  def rq_gripper_led_force_blue(gripper_socket="1"):
      rq_set_var(LBP,1, gripper_socket)
      rq_set_var(LRD,0, gripper_socket)
      rq_set_var(LBL,1, gripper_socket)
      rq_set_var(LGN,0, gripper_socket)
  end

  def rq_gripper_led_force_green(gripper_socket="1"):
      rq_set_var(LBP,1, gripper_socket)
      rq_set_var(LRD,0, gripper_socket)
      rq_set_var(LBL,0, gripper_socket)
      rq_set_var(LGN,1, gripper_socket)
  end

  def rq_gripper_led_force_purple(gripper_socket="1"):
      rq_set_var(LBP,1, gripper_socket)
      rq_set_var(LRD,1, gripper_socket)
      rq_set_var(LBL,1, gripper_socket)
      rq_set_var(LGN,0, gripper_socket)
  end

  ############################################
  # mm/inches functions
  ############################################
  gripper_closed_norm = [100, 100, 100, 100]
  gripper_open_norm = [0, 0, 0, 0]
  gripper_closed_mm = [0, 0, 0, 0]
  gripper_open_mm = [50, 50, 50, 50]

  def rq_current_pos_mm(gripper_socket=1):
      pos_gripper = rq_current_pos(gripper_socket)
      pos_mm = gripper_to_mm(pos_gripper, gripper_socket)
      return round_value_2_dec(pos_mm)
  end

  def rq_current_pos_inches(gripper_socket=1):
      pos_gripper = rq_current_pos(gripper_socket)
      pos_mm = gripper_to_mm(pos_gripper, gripper_socket)
      pos_in = pos_mm / 25.4
      return round_value_2_dec(pos_in)
  end

  def rq_move_mm(pos_mm, gripper_socket=1):
      pos_gripper = mm_to_gripper(pos_mm, gripper_socket)
      rq_move(pos_gripper, gripper_socket)
  end

  def rq_move_and_wait_mm(pos_mm, gripper_socket=1):
      pos_gripper = mm_to_gripper(pos_mm, gripper_socket)
      rq_move_and_wait(pos_gripper, gripper_socket)
  end

  def rq_move_inches(pos_in, gripper_socket=1):
      pos_mm = pos_in * 25.4
      rq_move_mm(pos_mm, gripper_socket)
  end

  def rq_move_and_wait_inches(pos_in, gripper_socket=1):
      pos_mm = pos_in * 25.4
      rq_move_and_wait_mm(pos_mm, gripper_socket)
  end

  def get_closed_norm(gripper_socket):
      return gripper_closed_norm[gripper_socket - 1]
  end

  def get_open_norm(gripper_socket):
      return gripper_open_norm[gripper_socket - 1]
  end

  def get_closed_mm(gripper_socket):
      return gripper_closed_mm[gripper_socket - 1]
  end

  def get_open_mm(gripper_socket):
      return gripper_open_mm[gripper_socket - 1]
  end

  def set_closed_norm(closed_norm, gripper_socket):
      gripper_closed_norm[gripper_socket - 1] = closed_norm
  end

  def set_open_norm(open_norm, gripper_socket):
      gripper_open_norm[gripper_socket - 1] = open_norm
  end

  def set_closed_mm(closed_mm, gripper_socket):
      gripper_closed_mm[gripper_socket - 1] = closed_mm
  end

  def set_open_mm(open_mm, gripper_socket):
      gripper_open_mm[gripper_socket - 1] = open_mm
  end

  def gripper_to_mm(value_gripper, gripper_socket):
      closed_norm = get_closed_norm(gripper_socket)
      open_norm = get_open_norm(gripper_socket)
      closed_mm = get_closed_mm(gripper_socket)
      open_mm = get_open_mm(gripper_socket)

      value_norm = (value_gripper / 255) * 100

      slope = (closed_mm - open_mm) / (closed_norm - open_norm)
      value_mm = slope * (value_norm - closed_norm) + closed_mm

      if (value_mm > open_mm):
          value_mm_limited = open_mm
      elif (value_mm < closed_mm):
          value_mm_limited = closed_mm
      else:
          value_mm_limited = value_mm
      end

      return value_mm_limited
  end

  def mm_to_gripper(value_mm, gripper_socket):
      closed_norm = get_closed_norm(gripper_socket)
      open_norm = get_open_norm(gripper_socket)
      closed_mm = get_closed_mm(gripper_socket)
      open_mm = get_open_mm(gripper_socket)

      slope = (closed_norm - open_norm) / (closed_mm - open_mm)
      value_norm = (value_mm - closed_mm) * slope + closed_norm

      value_gripper = value_norm * 255 / 100

      if (value_gripper > 255):
          value_gripper_limited = 255
      elif (value_gripper < 0):
          value_gripper_limited = 0
      else:
          value_gripper_limited = round_value(value_gripper)
      end

      return value_gripper_limited
  end

  def round_value(value):
      value_mod = value % 1

      if(value_mod < 0.5):
          return floor(value)
      else:
          return ceil(value)
      end
  end

  def round_value_2_dec(value):
      value_x_100 = value * 100
      value_x_100_rounded = round_value(value_x_100)
      return value_x_100_rounded / 100
  end

  def clear_socket_buffer(gripper_socket="1", read_timeout = 0.1):
    byte_in_buffer = socket_read_byte_list(1, gripper_socket, read_timeout)

    while(byte_in_buffer[0] >= 1):
        byte_in_buffer = socket_read_byte_list(1, gripper_socket, read_timeout)
    end
  end

  def rq_set_gripper_socket_acquire_option(enabled=False):
      gripper_socket_acquire_option = enabled

      if(not enabled):
          gripper_1_socket_acquired = False
          gripper_2_socket_acquired = False
          gripper_3_socket_acquired = False
          gripper_4_socket_acquired = False
      end
  end

  def rq_acquire_gripper_socket(gripper_socket="1"):
      if(gripper_socket_acquire_option):
          rq_wait_gripper_socket_released(gripper_socket)
          enter_critical
              rq_set_gripper_socket_acquired(gripper_socket, True)
          exit_critical

          clear_socket_buffer(gripper_socket, 0.002)

          sync()
      end
  end

  def rq_release_gripper_socket(gripper_socket="1"):
      if(gripper_socket_acquire_option):
          rq_set_gripper_socket_acquired(gripper_socket, False)

          sync()
      end
  end

  def rq_set_gripper_socket_acquired(gripper_socket="1", acquired=False):
      if(gripper_socket == "1"):
          gripper_1_socket_acquired = acquired
      elif(gripper_socket == "2"):
          gripper_2_socket_acquired = acquired
      elif(gripper_socket == "3"):
          gripper_3_socket_acquired = acquired
      elif(gripper_socket == "4"):
          gripper_4_socket_acquired = acquired
      end
  end

  def rq_get_gripper_socket_acquired(gripper_socket="1"):
      if(gripper_socket == "1"):
          return gripper_1_socket_acquired
      elif(gripper_socket == "2"):
          return gripper_2_socket_acquired
      elif(gripper_socket == "3"):
          return gripper_3_socket_acquired
      elif(gripper_socket == "4"):
          return gripper_4_socket_acquired
      end

      sync()
  end

  def rq_wait_gripper_socket_released(gripper_socket="1"):
      while(rq_get_gripper_socket_acquired(gripper_socket)):
          sync()
      end

      sync()
  end

  def scale(value, rawRange, scaledRange):
      def computeSlope(inputRange, outputRange):
          outputRangeDelta = outputRange[1] - outputRange[0]
          inputRangeDelta = inputRange[1] - inputRange[0]

          if (inputRangeDelta == 0):
              return 0
          else:
              return outputRangeDelta / inputRangeDelta
          end
      end

      def computeIntercept(slope, inputRange, outputRange):
          return outputRange[0] - (slope * inputRange[0])
      end

      def clipScaledValue(outputScaledValue, outputRange):
          if (outputRange[0] < outputRange[1]):
              return clipWhenLowerLimitIsLessThanHigher(outputScaledValue, outputRange)
          else:
              return clipWhenLowerLimitIsGreaterThanHigherLimit(outputScaledValue, outputRange)
          end
      end

      def clipWhenLowerLimitIsGreaterThanHigherLimit(outputScaledValue, outputRange):
          if (outputScaledValue < outputRange[1]):
              return outputRange[1]
          elif (outputScaledValue > outputRange[0]):
              return outputRange[0]
          else:
              return outputScaledValue
          end
      end

      def clipWhenLowerLimitIsLessThanHigher(outputScaledValue, outputRange):
          if (outputScaledValue < outputRange[0]):
              return outputRange[0]
          elif (outputScaledValue > outputRange[1]):
              return outputRange[1]
          else:
              return outputScaledValue
          end
      end

      slope = computeSlope(rawRange, scaledRange)
      intercept = computeIntercept(slope, rawRange, scaledRange)
      scaledValue = slope * value + intercept
      return clipScaledValue(scaledValue, scaledRange)
  end

  def limit(value, range):
      return scale(value, range, range)
  end


  rq_obj_detect = 0
  rq_init_comm_if_connected(9, "1")
  rq_init_comm_if_connected(2, "2")
  rq_init_comm_if_connected(3, "3")
  rq_init_comm_if_connected(4, "4")
  rq_print_connected_grippers()
  connectivity_checked = [-1,-1,-1,-1]
  status_checked = [-1,-1,-1,-1]
  current_speed = [-1,-1,-1,-1]
  current_force = [-1,-1,-1,-1]
  set_closed_norm(100.0, 1)
  set_open_norm(0.0, 1)
  set_closed_mm(0.0, 1)
  set_open_mm(50.0, 1)
  set_closed_norm(100.0, 2)
  set_open_norm(0.0, 2)
  set_closed_mm(0.0, 2)
  set_open_mm(50.0, 2)
  set_closed_norm(100.0, 3)
  set_open_norm(0.0, 3)
  set_closed_mm(0.0, 3)
  set_open_mm(50.0, 3)
  set_closed_norm(100.0, 4)
  set_open_norm(0.0, 4)
  set_closed_mm(0.0, 4)
  set_open_mm(50.0, 4)
  # end: URCap Installation Node
  $ 1 "BeforeStart"
  $ 2 "var_1≔ False "
  global var_1=  False
  $ 3 "thread_flag≔ False "
  global thread_flag=  False
  $ 4 "thread_var2≔0"
  global thread_var2=0
  $ 5 "var_10≔[0,0,0,0,0,0,0,0,0,0]"
  global var_10=[0,0,0,0,0,0,0,0,0,0]
  $ 6 "var_15≔ False "
  global var_15=  False
  $ 7 "Set CO[0]= False "
  set_configurable_digital_out(0,   False  )
  $ 8 "Set"
  set_tcp(p[0.0,0.0,0.11,0.0,0.0,0.0])
  $ 221 "Thread_1"
  thread Thread_1():
    while (True):
      $ 222 "Loop thread_flag== False "
      while (thread_flag==  False  ):
        $ 223 "var_12=0"
        var_12=0
        $ 224 "Wait: 0.01"
        sleep(0.01)
      end
      $ 225 "Wait: 0.001"
      sleep(0.001)
      $ 226 "var_11≔get_tcp_force()"
      global var_11=get_tcp_force()
      $ 227 "If var_11[axis]*var_11[axis]<var_2[11]*var_2[11]"
      if (var_11[axis]*var_11[axis]<var_2[11]*var_2[11]):
        $ 228 "var_12=0"
        var_12=0
      else:
        $ 229 "Else"
        $ 230 "var_12=var_12+1"
        var_12=var_12+1
        $ 231 "If var_12>0"
        if (var_12>0):
          $ 232 "thread_flag= False "
          thread_flag=  False
        end
      end
    end
  end
  threadId_Thread_1 = run Thread_1()
  $ 235 "Thread_2"
  thread Thread_2():
    while (True):
      $ 236 "Loop thread_var2==0"
      while (thread_var2==0):
        $ 237 "Wait: 0.01"
        sleep(0.01)
      end
      $ 238 "sleep(thread_var2)"
      sleep(thread_var2)
      $ 239 "var_5≔get_actual_tcp_pose()"
      global var_5=get_actual_tcp_pose()
      $ 240 "socket_send_string(var_5)"
      socket_send_string(var_5)
    end
  end
  threadId_Thread_2 = run Thread_2()
  thread EventThread():
    while (True):
      if (get_configurable_digital_in(0)):
        $ 242 "var_15= not var_15"
        var_15=  not  var_15
        $ 243 "Set CO[0]=var_15"
        set_configurable_digital_out(0, var_15)
        $ 244 "Wait: 0.3"
        sleep(0.3)
      end
      sync()
    end
  end
  eventThread = run EventThread()
  while (True):
    $ 9 "Robot Program"
    $ 10 "Loop var_1==False"
    while (var_1==False):
      $ 11 "var_1≔socket_open('192.168.1.5',30010)"
      global var_1=socket_open("192.168.1.5",30010)
      $ 12 "Wait: 0.5"
      sleep(0.5)
    end
    $ 13 "Loop var_1== True "
    thread Thread_while_13():
      while (True):
        $ 14 "Wait: 0.001"
        sleep(0.001)
        $ 15 "var_2≔socket_read_ascii_float(12)"
        global var_2=socket_read_ascii_float(12)
        $ 16 "Loop var_2[0]≠12"
        while (var_2[0] != 12):
          $ 17 "var_2≔socket_read_ascii_float(12)"
          global var_2=socket_read_ascii_float(12)
        end
        $ 18 "Switch var_2[1]"
        switch_1 = var_2[1]
        $ 19 "Case 0"
        if (0 == switch_1):
          $ 20 "'movejl'"
          # 'movejl'
          $ 21 "var_3≔p[var_2[2],var_2[3],var_2[4],var_2[5],var_2[6],var_2[7]]"
          global var_3=p[var_2[2],var_2[3],var_2[4],var_2[5],var_2[6],var_2[7]]
          $ 22 "movej(var_3,var_2[8],var_2[9],var_2[10],var_2[11])"
          movej(var_3,var_2[8],var_2[9],var_2[10],var_2[11])
          $ 23 "If var_2[12]==0"
          if (var_2[12]==0):
            $ 24 "socket_send_string('1')"
            socket_send_string("1")
          end
        elif (1 == switch_1):
          $ 25 "Case 1"
          $ 26 "'movej'"
          # 'movej'
          $ 27 "var_6≔[var_2[2],var_2[3],var_2[4],var_2[5],var_2[6],var_2[7]]"
          global var_6=[var_2[2],var_2[3],var_2[4],var_2[5],var_2[6],var_2[7]]
          $ 28 "movej(var_6,var_2[8],var_2[9],var_2[10],var_2[11])"
          movej(var_6,var_2[8],var_2[9],var_2[10],var_2[11])
          $ 29 "If var_2[12]==0"
          if (var_2[12]==0):
            $ 30 "socket_send_string('completed_joint_move')"
            socket_send_string("completed_joint_move")
          end
        elif (2 == switch_1):
          $ 31 "Case 2"
          $ 32 "'movel'"
          # 'movel'
          $ 33 "var_3≔p[var_2[2],var_2[3],var_2[4],var_2[5],var_2[6],var_2[7]]"
          global var_3=p[var_2[2],var_2[3],var_2[4],var_2[5],var_2[6],var_2[7]]
          $ 34 "movel(var_3,var_2[8],var_2[9],var_2[10],var_2[11])"
          movel(var_3,var_2[8],var_2[9],var_2[10],var_2[11])
          $ 35 "If var_2[12]==0"
          if (var_2[12]==0):
            $ 36 "socket_send_string('completed_linear_move')"
            socket_send_string("completed_linear_move")
          end
        elif (3 == switch_1):
          $ 37 "Case 3"
          $ 38 "'move to var_3 relative to current pose'"
          # 'move to var_3 relative to current pose'
          $ 39 "var_3≔p[var_2[2],var_2[3],var_2[4],var_2[5],var_2[6],var_2[7]]"
          global var_3=p[var_2[2],var_2[3],var_2[4],var_2[5],var_2[6],var_2[7]]
          $ 40 "var_5≔get_actual_tcp_pose()"
          global var_5=get_actual_tcp_pose()
          $ 41 "movel(pose_trans(var_5,var_3),var_2[8],var_2[9],var_2[10],var_2[11])"
          movel(pose_trans(var_5,var_3),var_2[8],var_2[9],var_2[10],var_2[11])
          $ 42 "If var_2[12]==0"
          if (var_2[12]==0):
            $ 43 "socket_send_string('completed_relative_linear_move')"
            socket_send_string("completed_relative_linear_move")
          end
        elif (4 == switch_1):
          $ 44 "Case 4"
          $ 45 "'force move in single axis'"
          # 'force move in single axis'
          $ 46 "var_5≔get_actual_tcp_pose()"
          global var_5=get_actual_tcp_pose()
          $ 47 "If var_2[2]≠0"
          if (var_2[2] != 0):
            $ 48 "var_5[0]=var_5[0]+var_2[2]"
            var_5[0]=var_5[0]+var_2[2]
            $ 49 "axis≔0"
            global axis=0
          else:
            $ 50 "ElseIf var_2[3]≠0"
            if (var_2[3] != 0):
              $ 51 "var_5[1]=var_5[1]+var_2[3]"
              var_5[1]=var_5[1]+var_2[3]
              $ 52 "axis≔1"
              global axis=1
            else:
              $ 53 "ElseIf var_2[4]≠0"
              if (var_2[4] != 0):
                $ 54 "var_5[2]=var_5[2]+var_2[4]"
                var_5[2]=var_5[2]+var_2[4]
                $ 55 "axis≔2"
                global axis=2
              end
            end
          end
          $ 56 "thread_flag= True "
          thread_flag=  True
          $ 57 "Loop thread_flag== True "
          thread Thread_while_57():
            while (True):
              $ 58 "movel(var_5,var_2[8],var_2[9],0,0)"
              movel(var_5,var_2[8],var_2[9],0,0)
              $ 59 "Wait: 0.01"
              sleep(0.01)
              $ 60 "thread_flag= False "
              thread_flag=  False
            end
          end
          if (thread_flag==  True  ):
            global thread_handler_57=run Thread_while_57()
            while (thread_flag==  True  ):
              sync()
            end
            kill thread_handler_57
          end
          $ 61 "stopl(10)"
          stopl(10)
          $ 62 "If var_2[12]==0"
          if (var_2[12]==0):
            $ 63 "socket_send_string('completed_force_move')"
            socket_send_string("completed_force_move")
          end
        elif (5 == switch_1):
          $ 64 "Case 5"
          $ 65 "'servoj'"
          # 'servoj'
          $ 66 "var_3≔p[var_2[2],var_2[3],var_2[4],var_2[5],var_2[6],var_2[7]]"
          global var_3=p[var_2[2],var_2[3],var_2[4],var_2[5],var_2[6],var_2[7]]
          $ 67 "If var_2[12]==0"
          if (var_2[12]==0):
            $ 68 "stopl(0.5)"
            stopl(0.5)
          else:
            $ 69 "Else"
            $ 70 "var_14≔get_inverse_kin(var_3)"
            global var_14=get_inverse_kin(var_3)
            $ 71 "servoj(var_14,t=var_2[9],lookahead_time=var_2[10],gain=var_2[11])"
            servoj(var_14,t=var_2[9],lookahead_time=var_2[10],gain=var_2[11])
          end
          $ 72 "If var_2[12]==0"
          if (var_2[12]==0):
            $ 73 "socket_send_string('completed_servoj_move')"
            socket_send_string("completed_servoj_move")
          end
        elif (6 == switch_1):
          $ 74 "Case 6"
          $ 75 "'speedl'"
          # 'speedl'
          $ 76 "var_6≔[var_2[2],var_2[3],var_2[4],var_2[5],var_2[6],var_2[7]]"
          global var_6=[var_2[2],var_2[3],var_2[4],var_2[5],var_2[6],var_2[7]]
          $ 77 "If var_2[10]==0"
          if (var_2[10]==0):
            $ 78 "speedl(var_6,var_2[8])"
            speedl(var_6,var_2[8])
          else:
            $ 79 "Else"
            $ 80 "speedl(var_6,var_2[8],var_2[10])"
            speedl(var_6,var_2[8],var_2[10])
          end
          $ 81 "socket_send_string('completed_speedl')"
          socket_send_string("completed_speedl")
        elif (7 == switch_1):
          $ 82 "Case 7"
          $ 83 "'speedj'"
          # 'speedj'
          $ 84 "var_6≔[var_2[2],var_2[3],var_2[4],var_2[5],var_2[6],var_2[7]]"
          global var_6=[var_2[2],var_2[3],var_2[4],var_2[5],var_2[6],var_2[7]]
          $ 85 "If var_2[10]==0"
          if (var_2[10]==0):
            $ 86 "speedj(var_6,var_2[8])"
            speedj(var_6,var_2[8])
          else:
            $ 87 "Else"
            $ 88 "speedj(var_6,var_2[8],var_2[10])"
            speedj(var_6,var_2[8],var_2[10])
          end
          $ 89 "socket_send_string('completed_speedj')"
          socket_send_string("completed_speedj")
        elif (8 == switch_1):
          $ 90 "Case 8"
          $ 91 "'stopl'"
          # 'stopl'
          $ 92 "stopl(var_2[8])"
          stopl(var_2[8])
          $ 93 "socket_send_string('completed_stopl')"
          socket_send_string("completed_stopl")
        elif (9 == switch_1):
          $ 94 "Case 9"
          $ 95 "'servoc'"
          # 'servoc'
          $ 96 "var_3≔p[var_2[2],var_2[3],var_2[4],var_2[5],var_2[6],var_2[7]]"
          global var_3=p[var_2[2],var_2[3],var_2[4],var_2[5],var_2[6],var_2[7]]
          $ 97 "If var_2[12]==0"
          if (var_2[12]==0):
            $ 98 "stopl(var_2[8])"
            stopl(var_2[8])
          else:
            $ 99 "Else"
            $ 100 "servoc(var_3,a=var_2[8],v=var_2[9],r=var_2[11])"
            servoc(var_3,a=var_2[8],v=var_2[9],r=var_2[11])
          end
          $ 101 "If var_2[12]==0"
          if (var_2[12]==0):
            $ 102 "socket_send_string('completed_servoc_move')"
            socket_send_string("completed_servoc_move")
          end
        elif (10 == switch_1):
          $ 103 "Case 10"
          $ 104 "'return current pose'"
          # 'return current pose'
          $ 105 "var_5≔get_actual_tcp_pose()"
          global var_5=get_actual_tcp_pose()
          $ 106 "socket_send_string(var_5)"
          socket_send_string(var_5)
        elif (11 == switch_1):
          $ 107 "Case 11"
          $ 108 "'return current joints'"
          # 'return current joints'
          $ 109 "var_4≔get_actual_joint_positions()"
          global var_4=get_actual_joint_positions()
          $ 110 "socket_send_string(var_4)"
          socket_send_string(var_4)
        elif (12 == switch_1):
          $ 111 "Case 12"
          $ 112 "'return inverse kin of pose'"
          # 'return inverse kin of pose'
          $ 113 "var_3≔p[var_2[2],var_2[3],var_2[4],var_2[5],var_2[6],var_2[7]]"
          global var_3=p[var_2[2],var_2[3],var_2[4],var_2[5],var_2[6],var_2[7]]
          $ 114 "socket_send_string(get_inverse_kin(var_3))"
          socket_send_string(get_inverse_kin(var_3))
        elif (13 == switch_1):
          $ 115 "Case 13"
          $ 116 "'return translation to get to 2nd pose from 1st pose coord system'"
          # 'return translation to get to 2nd pose from 1st pose coord system'
          $ 117 "var_3≔p[var_2[2],var_2[3],var_2[4],var_2[5],var_2[6],var_2[7]]"
          global var_3=p[var_2[2],var_2[3],var_2[4],var_2[5],var_2[6],var_2[7]]
          $ 118 "var_5≔get_actual_tcp_pose()"
          global var_5=get_actual_tcp_pose()
          $ 119 "socket_send_string(pose_trans(var_5,var_3))"
          socket_send_string(pose_trans(var_5,var_3))
        elif (14 == switch_1):
          $ 120 "Case 14"
          $ 121 "'return current forces'"
          # 'return current forces'
          $ 122 "socket_send_string(get_tcp_force())"
          socket_send_string(get_tcp_force())
        elif (15 == switch_1):
          $ 123 "Case 15"
          $ 124 "'return force magnitude'"
          # 'return force magnitude'
          $ 125 "socket_send_string(force())"
          socket_send_string(force())
        elif (16 == switch_1):
          $ 126 "Case 16"
          $ 127 "'return tool velocity'"
          # 'return tool velocity'
          $ 128 "socket_send_string(get_actual_tcp_speed())"
          socket_send_string(get_actual_tcp_speed())
        elif (17 == switch_1):
          $ 129 "Case 17"
          $ 130 "'return force magnitude'"
          # 'return force magnitude'
          $ 131 "socket_send_string(get_actual_joint_speeds())"
          socket_send_string(get_actual_joint_speeds())
        elif (18 == switch_1):
          $ 132 "Case 18"
          $ 133 "'return special tool state'"
          # 'return special tool state'
          $ 134 "socket_send_string(var_15)"
          socket_send_string(var_15)
        elif (19 == switch_1):
          $ 135 "Case 19"
          $ 136 "'return translation to get to 2nd pose from 1st pose coord system'"
          # 'return translation to get to 2nd pose from 1st pose coord system'
          $ 137 "var_3≔p[var_2[2],var_2[3],var_2[4],var_2[5],var_2[6],var_2[7]]"
          global var_3=p[var_2[2],var_2[3],var_2[4],var_2[5],var_2[6],var_2[7]]
          $ 139 "socket_send_string(pose_inv(var_3))"
          socket_send_string(pose_inv(var_3))
        elif (20 == switch_1):
          $ 140 "Case 20"
          $ 141 "'set tcp'"
          # 'set tcp'
          $ 142 "var_3≔p[var_2[2],var_2[3],var_2[4],var_2[5],var_2[6],var_2[7]]"
          global var_3=p[var_2[2],var_2[3],var_2[4],var_2[5],var_2[6],var_2[7]]
          $ 143 "set_tcp(var_3)"
          set_tcp(var_3)
          $ 144 "If var_2[12]==0"
          if (var_2[12]==0):
            $ 145 "socket_send_string('tcp_updated')"
            socket_send_string("tcp_updated")
          end
        elif (21 == switch_1):
          $ 146 "Case 21"
          $ 147 "'set payload'"
          # 'set payload'
          $ 148 "set_payload(var_2[8],[var_2[2],var_2[3],var_2[4]])"
          set_payload(var_2[8],[var_2[2],var_2[3],var_2[4]])
          $ 149 "If var_2[12]==0"
          if (var_2[12]==0):
            $ 150 "socket_send_string('payload_updated')"
            socket_send_string("payload_updated")
          end
        elif (22 == switch_1):
          $ 151 "Case 22"
          $ 152 "'set digital out'"
          # 'set digital out'
          $ 153 "If var_2[9]==1"
          if (var_2[9]==1):
            $ 154 "set_configurable_digital_out(var_2[8], True )"
            set_configurable_digital_out(var_2[8],  True  )
            $ 155 "If var_2[8]==0"
            if (var_2[8]==0):
              $ 156 "var_15= True "
              var_15=  True
              $ 157 "Set CO[0]= True "
              set_configurable_digital_out(0,   True  )
            end
          else:
            $ 158 "Else"
            $ 159 "set_configurable_digital_out(var_2[8], False )"
            set_configurable_digital_out(var_2[8],  False  )
            $ 160 "If var_2[8]==0"
            if (var_2[8]==0):
              $ 161 "var_15= False "
              var_15=  False
              $ 162 "Set CO[0]= False "
              set_configurable_digital_out(0,   False  )
            end
          end
          $ 163 "If var_2[12]==0"
          if (var_2[12]==0):
            $ 164 "socket_send_string('digital_output_set')"
            socket_send_string("digital_output_set")
          end
        elif (30 == switch_1):
          $ 165 "Case 30"
          $ 166 "freedrive_mode()"
          freedrive_mode()
          $ 167 "socket_send_string('begin_freedrive_mode')"
          socket_send_string("begin_freedrive_mode")
        elif (31 == switch_1):
          $ 168 "Case 31"
          $ 169 "end_freedrive_mode()"
          end_freedrive_mode()
          $ 170 "socket_send_string('end_freedrive_mode')"
          socket_send_string("end_freedrive_mode")
        elif (32 == switch_1):
          $ 171 "Case 32"
          $ 172 "socket_send_string('begin_blend_move')"
          socket_send_string("begin_blend_move")
          $ 173 "var_13≔var_2[8]"
          global var_13=var_2[8]
          $ 174 "n≔0"
          global n=0
          $ 175 "Loop n<var_13"
          while (n<var_13):
            $ 176 "n=n+1"
            n=n+1
            $ 177 "Loop var_2[0]≠12"
            while (var_2[0] != 12):
              $ 178 "var_2≔socket_read_ascii_float(12)"
              global var_2=socket_read_ascii_float(12)
            end
            $ 179 "var_3≔p[var_2[2],var_2[3],var_2[4],var_2[5],var_2[6],var_2[7]]"
            global var_3=p[var_2[2],var_2[3],var_2[4],var_2[5],var_2[6],var_2[7]]
            $ 180 "var_10[n] = var_3"
            var_10[n] = var_3
          end
          $ 181 "movel(var_10[0],0.1,0.5,0,0)"
          movel(var_10[0],0.1,0.5,0,0)
          $ 182 "n≔0"
          global n=0
          $ 183 "Loop n<var_13"
          while (n<var_13):
            $ 184 "n=n+1"
            n=n+1
            $ 185 "movep(var_10[n])"
            movep(var_10[n])
          end
        elif (33 == switch_1):
          $ 186 "Case 33"
          $ 187 "socket_send_string('begin_blend_move')"
          socket_send_string("begin_blend_move")
        elif (40 == switch_1):
          $ 188 "Case 40"
          $ 189 "socket_send_string('robot_ready')"
          socket_send_string("robot_ready")
        elif (41 == switch_1):
          $ 190 "Case 41"
          $ 191 "thread_var2=var_2[8]"
          thread_var2=var_2[8]
          $ 192 "socket_send_string('data_streaming_started')"
          socket_send_string("data_streaming_started")
        elif (42 == switch_1):
          $ 193 "Case 42"
          $ 194 "thread_var2=0"
          thread_var2=0
          $ 195 "socket_send_string('data_streaming_stopped')"
          socket_send_string("data_streaming_stopped")
        elif (100 == switch_1):
          $ 196 "Case 100"
          $ 197 "'reset program'"
          # 'reset program'
          $ 198 "If var_2[12]==0"
          if (var_2[12]==0):
            $ 199 "socket_send_string('resetting...')"
            socket_send_string("resetting...")
          end
          $ 200 "socket_close()"
          socket_close()
          $ 201 "var_1≔ False "
          global var_1=  False
        elif (101 == switch_1):
          $ 202 "Case 101"
          $ 203 "socket_send_string('ready')"
          socket_send_string("ready")
        elif (400 == switch_1):
          $ 204 "Case 400"
          $ 205 "'safe move'"
          # 'safe move'
          $ 206 "var_3≔p[var_2[2],var_2[3],var_2[4],var_2[5],var_2[6],var_2[7]]"
          global var_3=p[var_2[2],var_2[3],var_2[4],var_2[5],var_2[6],var_2[7]]
          $ 207 "var_5≔get_actual_tcp_pose()"
          global var_5=get_actual_tcp_pose()
          $ 208 "var_7≔get_inverse_kin(var_3)"
          global var_7=get_inverse_kin(var_3)
          $ 209 "var_8≔get_inverse_kin(var_5)"
          global var_8=get_inverse_kin(var_5)
          $ 210 "var_9≔0"
          global var_9=0
          $ 211 "Loop 6 times"
          Loop_5 = 0
          while (Loop_5 < 6):
            $ 212 "If (var_7[Loop_5]-var_8[Loop_5])>2.0  or  (var_8[Loop_5]-var_7[Loop_5])>2.0"
            if ((var_7[Loop_5]-var_8[Loop_5])>2.0   or   (var_8[Loop_5]-var_7[Loop_5])>2.0):
              $ 213 "var_9=1"
              var_9=1
            end
            Loop_5 = Loop_5 + 1
          end
          $ 215 "If var_9==0"
          if (var_9==0):
            $ 216 "movej(var_3,1,var_2[8],0,0)"
            movej(var_3,1,var_2[8],0,0)
            $ 217 "socket_send_string('completed_pose_move')"
            socket_send_string("completed_pose_move")
          else:
            $ 218 "Else"
            $ 219 "socket_send_string('no_safe_move_found')"
            socket_send_string("no_safe_move_found")
          end
        end
      end
    end
    if (var_1==  True  ):
      global thread_handler_13=run Thread_while_13()
      while (var_1==  True  ):
        sync()
      end
      kill thread_handler_13
    end
  end
end
